TYPE PositionExtremaDesc :
STRUCT
  Minimum, Maximum : LREAL;
  Tmin, Tmax : LREAL;  
END_STRUCT
END_TYPE

(* stored: Version 1.1.0.1, ProductVersion 3.1.4024.9
   DUT PositionExtremaDesc: Id {b615dcba-8544-436f-9a57-30985945064e} *)
